INTERFACE I_Base EXTENDS __SYSTEM.IQueryInterface

METHOD Base : BOOL
VAR_INPUT
END_VAR
END_METHOD

END_INTERFACE

(* stored: Version 1.1.0.1, ProductVersion 3.1.4024.12
   Itf I_Base: Id {737d8c2f-a30e-4e95-9295-d6a8108b5747}
   Method Base: Id {87bdf4b9-4780-481f-938c-afb6ee294d86} *)
